Staubli VAL3: typeLen.pgx

public program typeLen(num pX, num pY, string pStr, num pLen)
begin
  //---------------------------------
  //  S H O W   O N E   S T R I N G
  //---------------------------------
  // Display one message with the same
  // number of characters.
  //
  //
  // See type()
  //         1234567890123456789012345678901234567890
  call strlength(pStr,pLen)
  call type(pX,pY,pStr)
end
